Staubli VAL3: onInsert.pgx

public program onInsert(string& x_sItem[])
  local num l_nSize
  local num i
  local string l_sEvent
  local num l_nKey
  local string l_sType
begin
  cls()
  call language:message(l_sEvent,64)
  call use:clear(0,13)
  call use:typeCenter(13,l_sEvent,40,true)
  x_sItem=""
  call use:setSizeList(19,0,19,11)
  call getType(l_sType)
  call use:listcreate(l_sType+" ")
  call getSize(l_nSize)
  if l_nSize!=0
    for i=0 to l_nSize-1
      call get(l_sEvent,i)
      call use:listadd(l_sEvent)
    endFor
    call use:listupdate(0)
    do
      l_nKey=get()
      call use:listevent(l_nKey,i,l_sEvent)
    until l_nKey==255 or l_nKey==270
    if l_nKey==270
      x_sItem=l_sEvent
    endIf
  endIf
  call use:nullKey(l_nKey)
end
